// TIA Portal V17 export
// export: Created 2026-04-13T11:12:44.0108649Z, ExportSetting WithDefaults, DisplayName Totally Integrated Automation Portal, DisplayVersion V17 Update 4, DisplayName TIA Portal Openness, DisplayVersion V17 Update 4, DisplayName TIA Portal Version Control Interface, DisplayVersion V17, DisplayName SINAMICS Startdrive Advanced, DisplayVersion V17, DisplayName SINAMICS Startdrive G130, G150, S120, S150, SINAMICS MV, S210, DisplayVersion V17, DisplayName SINAMICS Startdrive G110M, G120, G120C, G120D, G120P, G115D, DisplayVersion V17, DisplayName STEP 7 Professional, DisplayVersion V17 Update 4, DisplayName STEP 7 Safety, DisplayVersion V17, DisplayName WinCC Professional, DisplayVersion V17 Update 4
FUNCTION_BLOCK "称重与流量"   // FB57, LAD
{ S7_Optimized_Access := 'FALSE' }
VERSION : 0.1
// stored: AutoNumber true, IsIECCheckEnabled false, SetENOAutomatically false, UDAEnableTagReadback false
   VAR_OUTPUT
      A瞬时流量 : Real;
      A瞬时流量AT AT A瞬时流量 : Array[0..1] of Word;
      A瞬时流速 : Real;
      A瞬时流速AT AT A瞬时流速 : Array[0..1] of Word;
      A当前电流 : Real;
      A当前电流AT AT A当前电流 : Array[0..1] of Word;
      A介质温度 : Real;
      A介质温度AT AT A介质温度 : Array[0..1] of Word;
      A当前采集 : Real;
      A当前采集AT AT A当前采集 : Array[0..1] of Word;
      A流速下限 : Real;
      A流速下限AT AT A流速下限 : Array[0..1] of Word;
      A流速上限 : Real;
      A流速上限AT AT A流速上限 : Array[0..1] of Word;
      A管道内径 : Real;
      A管道内径AT AT A管道内径 : Array[0..1] of Word;
      B瞬时流量 : Real;
      B瞬时流量AT AT B瞬时流量 : Array[0..1] of Word;
      B瞬时流速 : Real;
      B瞬时流速AT AT B瞬时流速 : Array[0..1] of Word;
      B当前电流 : Real;
      B当前电流AT AT B当前电流 : Array[0..1] of Word;
      B介质温度 : Real;
      B介质温度AT AT B介质温度 : Array[0..1] of Word;
      B当前采集 : Real;
      B当前采集AT AT B当前采集 : Array[0..1] of Word;
      B流速下限 : Real;
      B流速下限AT AT B流速下限 : Array[0..1] of Word;
      B流速上限 : Real;
      B流速上限AT AT B流速上限 : Array[0..1] of Word;
      B管道内径 : Real;
      B管道内径AT AT B管道内径 : Array[0..1] of Word;
   END_VAR
   VAR_IN_OUT
      "秤操作-去皮" : Bool;
      读重量 : Real;
   END_VAR
   VAR DB_SPECIFIC
      CTU { S7_SetPoint := 'True'} : CTU_INT;
      TEMP { S7_SetPoint := 'True'} : Bool;
      TON1 : TON_TIME;
      TP : Array[0..40] of Bool;
      秤操作辅助 : Int;
      CZTFZ : Int;
   END_VAR
   VAR
      CZT AT CZTFZ : Array[0..15] of Bool;
   END_VAR
   VAR DB_SPECIFIC
      ST1 : Array[0..5] of Word;
      ST2 : Array[0..7] of Word;
      ST3 : Array[0..1] of Word;
      ST4 : Array[0..5] of Word;
      ST5 : Array[0..7] of Word;
      ST6 : Array[0..1] of Word;
      ST7 : Array[0..1] of Word;
      读重量辅助 : DInt;
   END_VAR
   VAR
      读重量辅助AT AT 读重量辅助 : Array[0..1] of Word;
      Modbus_Comm_Load { S7_SetPoint := 'True'} : Modbus_Comm_Load;
      Modbus_Master { S7_SetPoint := 'True'} : Modbus_Master;
   END_VAR
   VAR_TEMP   // added for the SCL form of the ladder/FBD networks
      _w1 : Bool;
      _w2 : Bool;
      _w3 : Bool;
   END_VAR
BEGIN

REGION Network 1
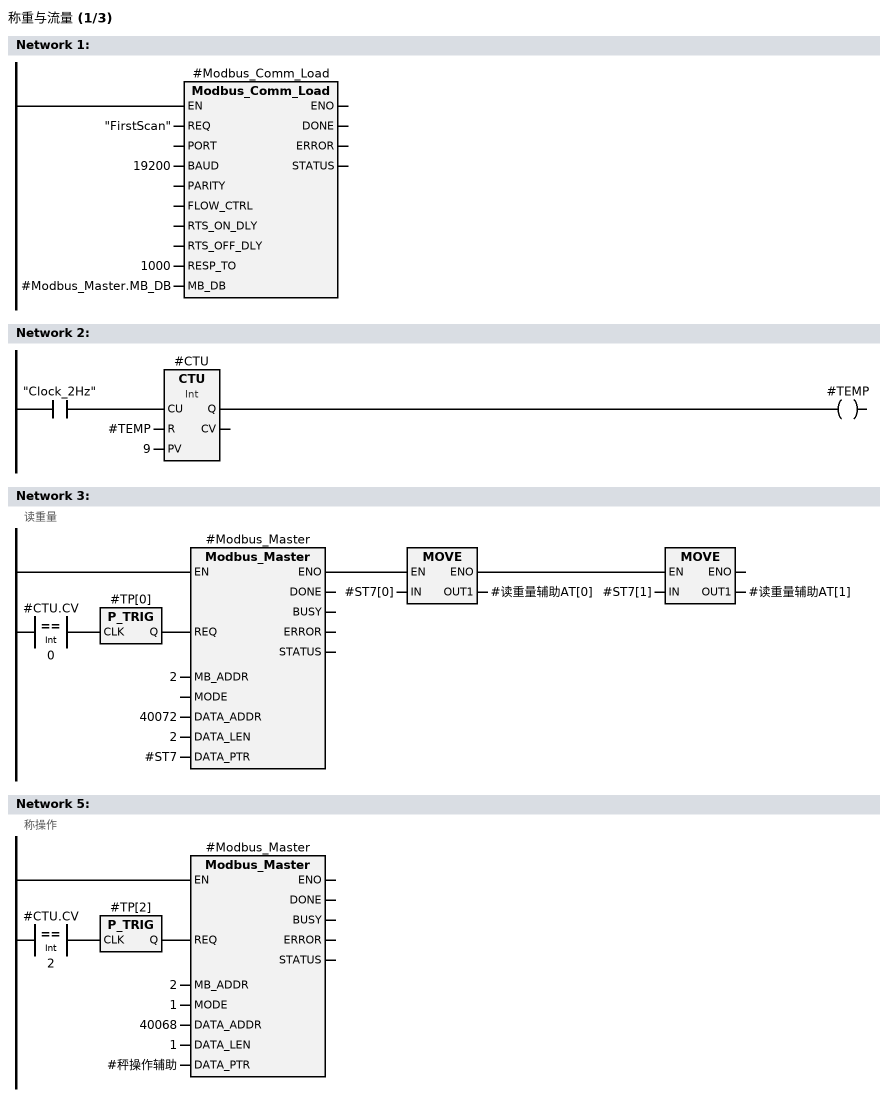
   RUNG wire#powerrail
      #Modbus_Comm_Load.Modbus_Comm_Load(REQ := "FirstScan", PORT :=, BAUD := 19200, PARITY :=, FLOW_CTRL :=, RTS_ON_DLY :=, RTS_OFF_DLY :=, RESP_TO := 1000, MB_DB := #Modbus_Master.MB_DB, DONE =>, ERROR =>, STATUS =>)
   END_RUNG
   // the same network as SCL:
   #Modbus_Comm_Load(REQ := "FirstScan", BAUD := 19200, RESP_TO := 1000, MB_DB := #Modbus_Master.MB_DB);   // Modbus_Comm_Load
END_REGION

REGION Network 2
   RUNG wire#powerrail
      Contact( "Clock_2Hz" )
      { S7_Templates := "value_type := Int" } #CTU.CTU(r := #TEMP, pv := 9, cv =>)
      Coil( #TEMP )
   END_RUNG
   // the same network as SCL:
   #CTU(CU := "Clock_2Hz", R := #TEMP, PV := 9);   // CTU
   #TEMP := #CTU.Q;
END_REGION

REGION Network 3
   // 读重量
   RUNG wire#powerrail
      #Modbus_Master.Modbus_Master(REQ := wire#w1, MB_ADDR := 2, MODE :=, DATA_ADDR := 40072, DATA_LEN := 2, DATA_PTR := #ST7, DONE =>, BUSY =>, ERROR =>, STATUS =>)
      Move(in := #ST7[0], out1 => #读重量辅助AT[0])
      Move(in := #ST7[1], out1 => #读重量辅助AT[1])
   END_RUNG
   RUNG wire#powerrail
      { S7_Templates := "SrcType := Int" } EQ_Contact(in1 := #CTU.CV, in2 := 0)
      P_Trig( #TP[0] )
   END_RUNG wire#w1
   // the same network as SCL:
   #_w1 := #CTU.CV = 0;
   #_w2 := #_w1 AND NOT #TP[0];   // rising edge
   #TP[0] := #_w1;
   #Modbus_Master(REQ := #_w2, MB_ADDR := 2, DATA_ADDR := 40072, DATA_LEN := 2, DATA_PTR := #ST7, ENO => #_w3);   // Modbus_Master
   IF #_w3 THEN
       #读重量辅助AT[0] := #ST7[0];
       #读重量辅助AT[1] := #ST7[1];
   END_IF;
END_REGION

REGION Network 4 (SCL)


   #读重量 := DINT_TO_REAL(#读重量辅助) * 0.01;
END_REGION

REGION Network 5
   // 称操作
   RUNG wire#powerrail
      #Modbus_Master.Modbus_Master(REQ := wire#w1, MB_ADDR := 2, MODE := 1, DATA_ADDR := 40068, DATA_LEN := 1, DATA_PTR := #秤操作辅助, DONE =>, BUSY =>, ERROR =>, STATUS =>)
   END_RUNG
   RUNG wire#powerrail
      { S7_Templates := "SrcType := Int" } EQ_Contact(in1 := #CTU.CV, in2 := 2)
      P_Trig( #TP[2] )
   END_RUNG wire#w1
   // the same network as SCL:
   #_w1 := #CTU.CV = 2;
   #_w2 := #_w1 AND NOT #TP[2];   // rising edge
   #TP[2] := #_w1;
   #Modbus_Master(REQ := #_w2, MB_ADDR := 2, MODE := 1, DATA_ADDR := 40068, DATA_LEN := 1, DATA_PTR := #秤操作辅助);   // Modbus_Master
END_REGION

REGION Network 6 (SCL)


   IF #"秤操作-去皮" = TRUE THEN
       #秤操作辅助 := 11;
       #"秤操作-去皮" := 0;

   END_IF;



   #TON1(IN := #秤操作辅助<>0,
         PT := T#5S);

   IF #TON1.Q THEN
       #秤操作辅助 := 0;

   END_IF;
END_REGION

REGION Network 7
   // 读流量
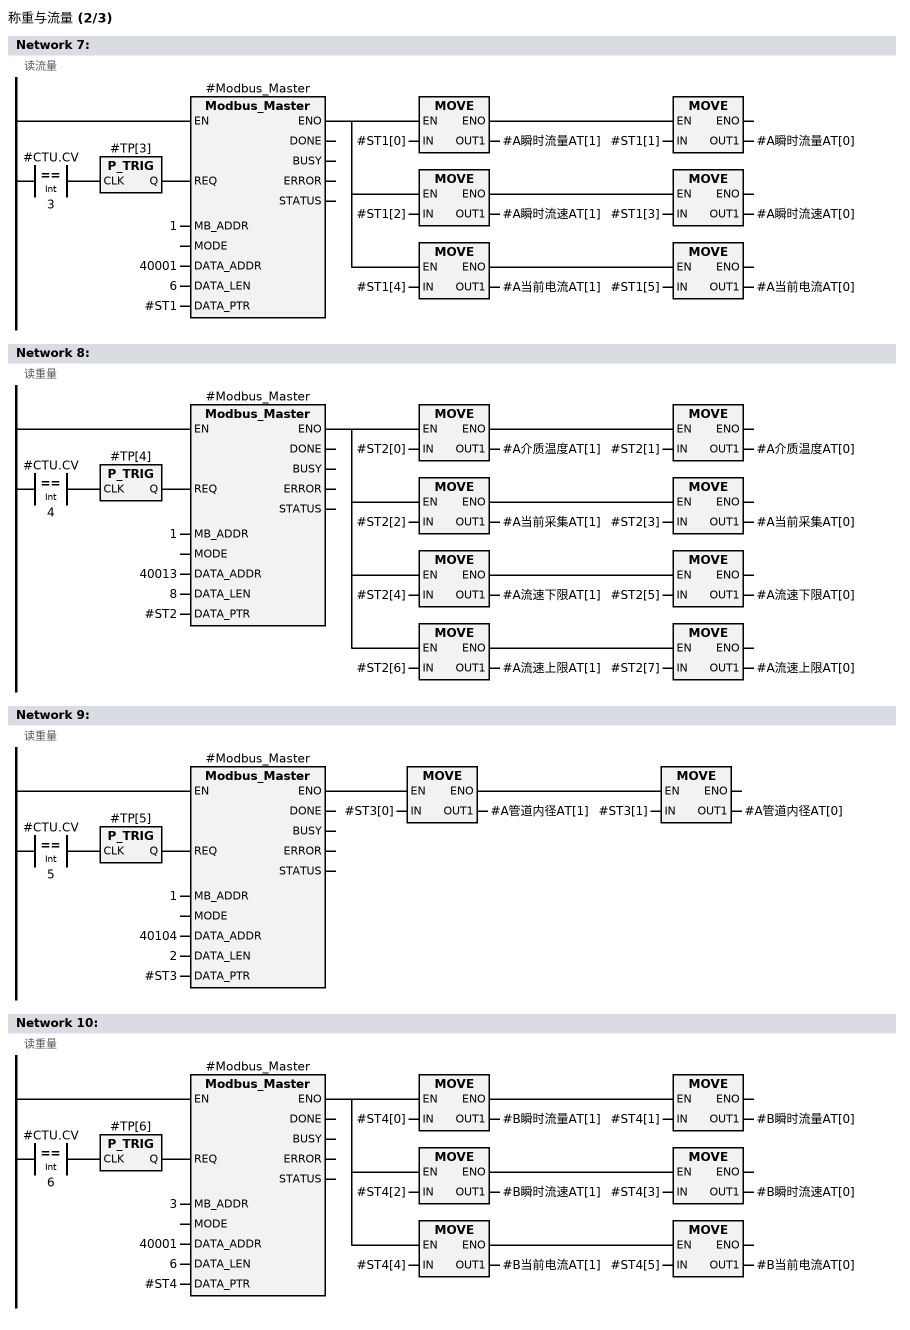
   RUNG wire#powerrail
      #Modbus_Master.Modbus_Master(REQ := wire#w1, MB_ADDR := 1, MODE :=, DATA_ADDR := 40001, DATA_LEN := 6, DATA_PTR := #ST1, DONE =>, BUSY =>, ERROR =>, STATUS =>)
      wire#w2
      Move(in := #ST1[0], out1 => #A瞬时流量AT[1])
      Move(in := #ST1[1], out1 => #A瞬时流量AT[0])
   END_RUNG
   RUNG wire#powerrail
      { S7_Templates := "SrcType := Int" } EQ_Contact(in1 := #CTU.CV, in2 := 3)
      P_Trig( #TP[3] )
   END_RUNG wire#w1
   RUNG wire#w2
      Move(in := #ST1[2], out1 => #A瞬时流速AT[1])
      Move(in := #ST1[3], out1 => #A瞬时流速AT[0])
   END_RUNG
   RUNG wire#w2
      Move(in := #ST1[4], out1 => #A当前电流AT[1])
      Move(in := #ST1[5], out1 => #A当前电流AT[0])
   END_RUNG
   // the same network as SCL:
   #_w1 := #CTU.CV = 3;
   #_w2 := #_w1 AND NOT #TP[3];   // rising edge
   #TP[3] := #_w1;
   #Modbus_Master(REQ := #_w2, MB_ADDR := 1, DATA_ADDR := 40001, DATA_LEN := 6, DATA_PTR := #ST1, ENO => #_w3);   // Modbus_Master
   IF #_w3 THEN
       #A瞬时流量AT[1] := #ST1[0];
       #A瞬时流量AT[0] := #ST1[1];
       #A瞬时流速AT[1] := #ST1[2];
       #A瞬时流速AT[0] := #ST1[3];
       #A当前电流AT[1] := #ST1[4];
       #A当前电流AT[0] := #ST1[5];
   END_IF;
END_REGION

REGION Network 8
   // 读重量
   RUNG wire#powerrail
      #Modbus_Master.Modbus_Master(REQ := wire#w1, MB_ADDR := 1, MODE :=, DATA_ADDR := 40013, DATA_LEN := 8, DATA_PTR := #ST2, DONE =>, BUSY =>, ERROR =>, STATUS =>)
      wire#w2
      Move(in := #ST2[0], out1 => #A介质温度AT[1])
      Move(in := #ST2[1], out1 => #A介质温度AT[0])
   END_RUNG
   RUNG wire#powerrail
      { S7_Templates := "SrcType := Int" } EQ_Contact(in1 := #CTU.CV, in2 := 4)
      P_Trig( #TP[4] )
   END_RUNG wire#w1
   RUNG wire#w2
      Move(in := #ST2[2], out1 => #A当前采集AT[1])
      Move(in := #ST2[3], out1 => #A当前采集AT[0])
   END_RUNG
   RUNG wire#w2
      Move(in := #ST2[4], out1 => #A流速下限AT[1])
      Move(in := #ST2[5], out1 => #A流速下限AT[0])
   END_RUNG
   RUNG wire#w2
      Move(in := #ST2[6], out1 => #A流速上限AT[1])
      Move(in := #ST2[7], out1 => #A流速上限AT[0])
   END_RUNG
   // the same network as SCL:
   #_w1 := #CTU.CV = 4;
   #_w2 := #_w1 AND NOT #TP[4];   // rising edge
   #TP[4] := #_w1;
   #Modbus_Master(REQ := #_w2, MB_ADDR := 1, DATA_ADDR := 40013, DATA_LEN := 8, DATA_PTR := #ST2, ENO => #_w3);   // Modbus_Master
   IF #_w3 THEN
       #A介质温度AT[1] := #ST2[0];
       #A介质温度AT[0] := #ST2[1];
       #A当前采集AT[1] := #ST2[2];
       #A当前采集AT[0] := #ST2[3];
       #A流速下限AT[1] := #ST2[4];
       #A流速下限AT[0] := #ST2[5];
       #A流速上限AT[1] := #ST2[6];
       #A流速上限AT[0] := #ST2[7];
   END_IF;
END_REGION

REGION Network 9
   // 读重量
   RUNG wire#powerrail
      #Modbus_Master.Modbus_Master(REQ := wire#w1, MB_ADDR := 1, MODE :=, DATA_ADDR := 40104, DATA_LEN := 2, DATA_PTR := #ST3, DONE =>, BUSY =>, ERROR =>, STATUS =>)
      Move(in := #ST3[0], out1 => #A管道内径AT[1])
      Move(in := #ST3[1], out1 => #A管道内径AT[0])
   END_RUNG
   RUNG wire#powerrail
      { S7_Templates := "SrcType := Int" } EQ_Contact(in1 := #CTU.CV, in2 := 5)
      P_Trig( #TP[5] )
   END_RUNG wire#w1
   // the same network as SCL:
   #_w1 := #CTU.CV = 5;
   #_w2 := #_w1 AND NOT #TP[5];   // rising edge
   #TP[5] := #_w1;
   #Modbus_Master(REQ := #_w2, MB_ADDR := 1, DATA_ADDR := 40104, DATA_LEN := 2, DATA_PTR := #ST3, ENO => #_w3);   // Modbus_Master
   IF #_w3 THEN
       #A管道内径AT[1] := #ST3[0];
       #A管道内径AT[0] := #ST3[1];
   END_IF;
END_REGION

REGION Network 10
   // 读重量
   RUNG wire#powerrail
      #Modbus_Master.Modbus_Master(REQ := wire#w1, MB_ADDR := 3, MODE :=, DATA_ADDR := 40001, DATA_LEN := 6, DATA_PTR := #ST4, DONE =>, BUSY =>, ERROR =>, STATUS =>)
      wire#w2
      Move(in := #ST4[0], out1 => #B瞬时流量AT[1])
      Move(in := #ST4[1], out1 => #B瞬时流量AT[0])
   END_RUNG
   RUNG wire#powerrail
      { S7_Templates := "SrcType := Int" } EQ_Contact(in1 := #CTU.CV, in2 := 6)
      P_Trig( #TP[6] )
   END_RUNG wire#w1
   RUNG wire#w2
      Move(in := #ST4[2], out1 => #B瞬时流速AT[1])
      Move(in := #ST4[3], out1 => #B瞬时流速AT[0])
   END_RUNG
   RUNG wire#w2
      Move(in := #ST4[4], out1 => #B当前电流AT[1])
      Move(in := #ST4[5], out1 => #B当前电流AT[0])
   END_RUNG
   // the same network as SCL:
   #_w1 := #CTU.CV = 6;
   #_w2 := #_w1 AND NOT #TP[6];   // rising edge
   #TP[6] := #_w1;
   #Modbus_Master(REQ := #_w2, MB_ADDR := 3, DATA_ADDR := 40001, DATA_LEN := 6, DATA_PTR := #ST4, ENO => #_w3);   // Modbus_Master
   IF #_w3 THEN
       #B瞬时流量AT[1] := #ST4[0];
       #B瞬时流量AT[0] := #ST4[1];
       #B瞬时流速AT[1] := #ST4[2];
       #B瞬时流速AT[0] := #ST4[3];
       #B当前电流AT[1] := #ST4[4];
       #B当前电流AT[0] := #ST4[5];
   END_IF;
END_REGION

REGION Network 11
   // 读重量
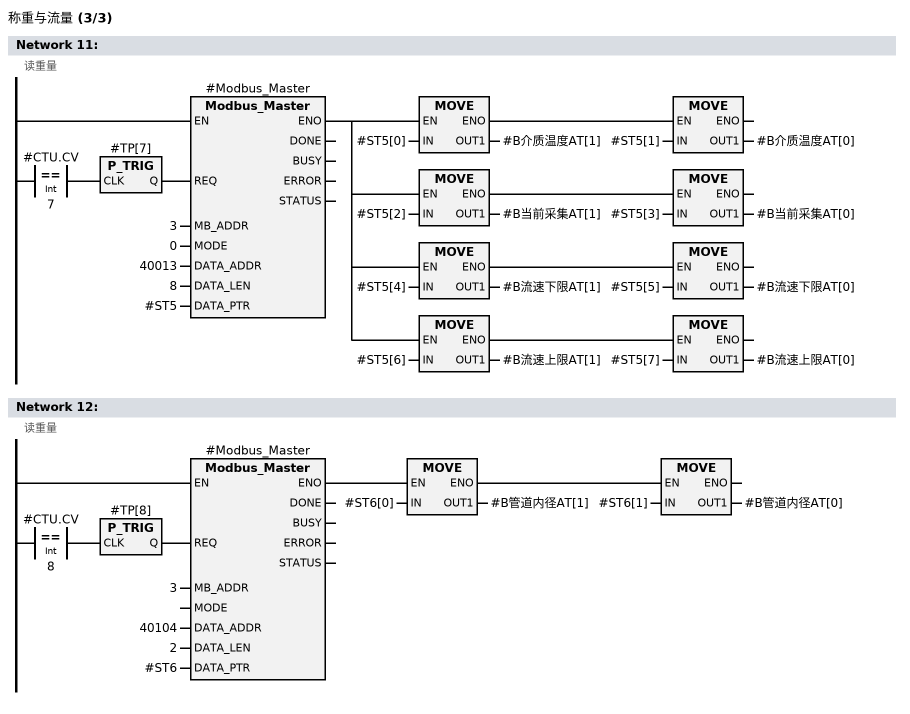
   RUNG wire#powerrail
      #Modbus_Master.Modbus_Master(REQ := wire#w1, MB_ADDR := 3, MODE := 0, DATA_ADDR := 40013, DATA_LEN := 8, DATA_PTR := #ST5, DONE =>, BUSY =>, ERROR =>, STATUS =>)
      wire#w2
      Move(in := #ST5[0], out1 => #B介质温度AT[1])
      Move(in := #ST5[1], out1 => #B介质温度AT[0])
   END_RUNG
   RUNG wire#powerrail
      { S7_Templates := "SrcType := Int" } EQ_Contact(in1 := #CTU.CV, in2 := 7)
      P_Trig( #TP[7] )
   END_RUNG wire#w1
   RUNG wire#w2
      Move(in := #ST5[2], out1 => #B当前采集AT[1])
      Move(in := #ST5[3], out1 => #B当前采集AT[0])
   END_RUNG
   RUNG wire#w2
      Move(in := #ST5[4], out1 => #B流速下限AT[1])
      Move(in := #ST5[5], out1 => #B流速下限AT[0])
   END_RUNG
   RUNG wire#w2
      Move(in := #ST5[6], out1 => #B流速上限AT[1])
      Move(in := #ST5[7], out1 => #B流速上限AT[0])
   END_RUNG
   // the same network as SCL:
   #_w1 := #CTU.CV = 7;
   #_w2 := #_w1 AND NOT #TP[7];   // rising edge
   #TP[7] := #_w1;
   #Modbus_Master(REQ := #_w2,   // Modbus_Master
                  MB_ADDR := 3,
                  MODE := 0,
                  DATA_ADDR := 40013,
                  DATA_LEN := 8,
                  DATA_PTR := #ST5,
                  ENO => #_w3);
   IF #_w3 THEN
       #B介质温度AT[1] := #ST5[0];
       #B介质温度AT[0] := #ST5[1];
       #B当前采集AT[1] := #ST5[2];
       #B当前采集AT[0] := #ST5[3];
       #B流速下限AT[1] := #ST5[4];
       #B流速下限AT[0] := #ST5[5];
       #B流速上限AT[1] := #ST5[6];
       #B流速上限AT[0] := #ST5[7];
   END_IF;
END_REGION

REGION Network 12
   // 读重量
   RUNG wire#powerrail
      #Modbus_Master.Modbus_Master(REQ := wire#w1, MB_ADDR := 3, MODE :=, DATA_ADDR := 40104, DATA_LEN := 2, DATA_PTR := #ST6, DONE =>, BUSY =>, ERROR =>, STATUS =>)
      Move(in := #ST6[0], out1 => #B管道内径AT[1])
      Move(in := #ST6[1], out1 => #B管道内径AT[0])
   END_RUNG
   RUNG wire#powerrail
      { S7_Templates := "SrcType := Int" } EQ_Contact(in1 := #CTU.CV, in2 := 8)
      P_Trig( #TP[8] )
   END_RUNG wire#w1
   // the same network as SCL:
   #_w1 := #CTU.CV = 8;
   #_w2 := #_w1 AND NOT #TP[8];   // rising edge
   #TP[8] := #_w1;
   #Modbus_Master(REQ := #_w2, MB_ADDR := 3, DATA_ADDR := 40104, DATA_LEN := 2, DATA_PTR := #ST6, ENO => #_w3);   // Modbus_Master
   IF #_w3 THEN
       #B管道内径AT[1] := #ST6[0];
       #B管道内径AT[0] := #ST6[1];
   END_IF;
END_REGION
END_FUNCTION_BLOCK
